Staubli VAL3: prog.pjx

--- prog.pjx ---
Parameters version=s7.2.1 stackSize=5000 millimeterUnit=true
Data file=prog.dtx

--- prog.dtx ---
public string eventi
